(* PLC project  *)

CONFIGURATION Servo_Parameter
END_CONFIGURATION
